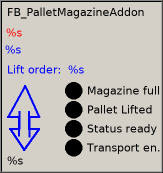
VISUALIZATION V_PalletMagazineAddon  // 163x173
VAR_IN_OUT
	{attribute 'VAR_IN_OUT_AS_POINTER'}
	fbFunction		: FB_PalletMagazineAddon;	
END_VAR
    Rectangle (0,0 163x173)
    Label (4,5 146x15), "FB_PalletMagazineAddon"
    Rectangle (4,151 104x20), "%s", text variable: fbFunction.ConfigFunction.FunctionName
    Rectangle (3,23 157x20), "%s", tooltip "%s", text variable: fbFunction.FunctionData.ErrorData.Error.ErrorCode.Conv, invisible if: fbFunction.FunctionData.ErrorData.Error.ErrorCode.Conv = 0
        p4168582468: fbFunction.FunctionData.ErrorData.Error.ErrorParam
    Rectangle (2,40 161x20), "%s", text variable: fbFunction.BaseFunctionData.States.eState
    Rectangle (4,60 155x20), "Lift order: %s", text variable: fbFunction.BaseFunctionData.OrderPosLift
    Polyline (19,136) (19,117) (8,117) (25,86) (39,117) (29,117) (29,137), invisible if: NOT fbFunction.HW_Outputs.LiftUp
    Polyline (19,111) (19,129) (10,129) (24,150) (39,129) (29,129) (29,111), invisible if: NOT fbFunction.HW_Outputs.LiftDown
    Ellipse (65,82 17x17), colour toggle: fbFunction.CtrlOut.MagazineFull
    Label (84,83 77x16), "Magazine full"
    Ellipse (65,101 17x17), colour toggle: fbFunction.CtrlOut.PalletLifted
    Label (84,102 77x16), "Pallet Lifted"
    Ellipse (65,120 17x17), colour toggle: fbFunction.CtrlOut.StatusReady
    Label (84,121 77x16), "Status ready"
    Ellipse (65,139 17x17), colour toggle: fbFunction.CtrlOut.TransportEnabled
    Label (84,140 77x16), "Transport en."
END_VISUALIZATION

(* stored: Version 1.1.0.1, ProductVersion 3.1.4024.9
   Visu V_PalletMagazineAddon: Id {d9a0cb84-5d06-49ef-9bf2-66cb3442af77} *)
